// TIA Portal V20 export
TYPE "typeCmControlNodeInterlock"
// stored: Namespace Unit1.Em2
   STRUCT
      jrOutPnPLeftAxisX : "LER_typeAxisInterlock";
      jrOutPnPLeftAxisZ : "LER_typeAxisInterlock";
      jrOutPnPRightAxisX : "LER_typeAxisInterlock";
      jrOutPnPRightAxisZ : "LER_typeAxisInterlock";
      jrOutPnPLeftClamp : "LER_typeTwoWayActuatorInterlock";
      jrOutPnPRightClamp : "LER_typeTwoWayActuatorInterlock";
   END_STRUCT;
END_TYPE
